FUNCTION_BLOCK ProxyControl (* Composite Function Block Type *)
  (* Standard: 61499-2 *)
  (* Version 0.0, 11/2/2016, chivdan, nxtControl GmbH, template *)
  PACKAGE Main;
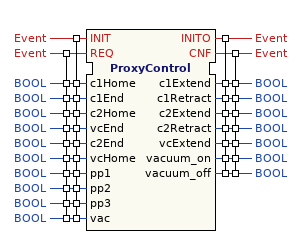
  EVENT_INPUT
    INIT WITH c1Home, c1End, c2Home, c2End, vcHome, vcEnd, pp1, pp2, pp3, vac; (* Initialization Request *)
    REQ WITH c1Home, c1End, c2Home, c2End, vcHome, vcEnd, pp1, pp2, pp3, vac; (* Normal Execution Request *)
  END_EVENT
  EVENT_OUTPUT
    INITO WITH c1Extend, c1Retract, c2Extend, c2Retract, vcExtend, vacuum_on, vacuum_off; (* Initialization Confirm *)
    CNF WITH c1Extend, c1Retract, c2Extend, c2Retract, vcExtend, vacuum_on, vacuum_off; (* Execution Confirmation *)
  END_EVENT
  VAR_INPUT
    c1Home : BOOL; (* Input event qualifier *)
    c1End : BOOL;
    c2Home : BOOL;
    vcEnd : BOOL;
    c2End : BOOL;
    vcHome : BOOL;
    pp1 : BOOL;
    pp2 : BOOL;
    pp3 : BOOL;
    vac : BOOL;
  END_VAR
  VAR_OUTPUT
    c1Extend : BOOL; (* Output event qualifier *)
    c1Retract : BOOL;
    c2Extend : BOOL;
    c2Retract : BOOL;
    vcExtend : BOOL;
    vacuum_on : BOOL;
    vacuum_off : BOOL;
  END_VAR
  FBS
    FB1 : CentralController;
    FB2 : InputLogger;
    FB3 : OutputLogger;
    FB4 : LogWriter;
  END_FBS
  EVENT_CONNECTIONS
    FB2.CNF TO FB1.REQ;
    FB2.INITO TO FB1.INIT;
    FB1.INITO TO FB3.INIT;
    FB3.INITO TO INITO;
    FB1.CNF TO FB3.REQ;
    FB3.CNF TO CNF;
    REQ TO FB2.REQ;
    INIT TO FB4.INIT;
    FB4.INITO TO FB2.INIT;
    FB2.WRITE_INPUT TO FB4.WRITE_INPUT;
    FB3.WRITE_OUTPUT TO FB4.WRITE_OUTPUT;
  END_CONNECTIONS
  DATA_CONNECTIONS
    c1Home TO FB2.x1;
    c1End TO FB2.x2;
    c2Home TO FB2.x3;
    c2End TO FB2.x4;
    vcHome TO FB2.x5;
    vcEnd TO FB2.x6;
    pp1 TO FB2.x7;
    pp2 TO FB2.x8;
    pp3 TO FB2.x9;
    vac TO FB2.x10;
    FB2.z1 TO FB1.c1Home;
    FB2.z2 TO FB1.c1End;
    FB2.z3 TO FB1.c2Home;
    FB2.z4 TO FB1.c2End;
    FB2.z5 TO FB1.vcHome;
    FB2.z6 TO FB1.vcEnd;
    FB2.z7 TO FB1.pp1;
    FB2.z8 TO FB1.pp2;
    FB2.z9 TO FB1.pp3;
    FB1.c1Extend TO FB3.x1;
    FB1.c1Retract TO FB3.x2;
    FB1.c2Extend TO FB3.x3;
    FB1.c2Retract TO FB3.x4;
    FB1.vcExtend TO FB3.x5;
    FB1.vacuum_on TO FB3.x6;
    FB1.vacuum_off TO FB3.x7;
    FB3.z1 TO c1Extend;
    FB3.z2 TO c1Retract;
    FB3.z3 TO c2Extend;
    FB3.z4 TO c2Retract;
    FB3.z5 TO vcExtend;
    FB3.z6 TO vacuum_on;
    FB3.z7 TO vacuum_off;
    FB2.z10 TO FB1.vac;
    FB2.z1 TO FB4.x1;
    FB2.z2 TO FB4.x2;
    FB2.z3 TO FB4.x3;
    FB2.z4 TO FB4.x4;
    FB2.z5 TO FB4.x5;
    FB2.z6 TO FB4.x6;
    FB2.z7 TO FB4.x7;
    FB2.z8 TO FB4.x8;
    FB2.z9 TO FB4.x9;
    FB2.z10 TO FB4.x10;
    FB3.z1 TO FB4.x11;
    FB3.z2 TO FB4.x12;
    FB3.z3 TO FB4.x13;
    FB3.z4 TO FB4.x14;
    FB3.z5 TO FB4.x15;
    FB3.z6 TO FB4.x16;
    FB3.z7 TO FB4.x17;
  END_CONNECTIONS
END_FUNCTION_BLOCK
